Staubli VAL3: action_suspend.pgx

program action_suspend()
begin
  // suspend all the task action
  if taskStatus("Cycle")!=-1
    taskSuspend("Cycle")
  endIf
  if taskStatus("Action")!=-1
    taskSuspend("Action")
  endIf
  //..

end
